KUKA KRL data list: Modul.dat

&ACCESS RVP
&REL 14
DEFDAT Modul PUBLIC
;FOLD EXTERNAL DECLARATIONS;%{PE}%MKUKATPBASIS,%CEXT,%VCOMMON,%P
;FOLD BASISTECH EXT;%{PE}%MKUKATPBASIS,%CEXT,%VEXT,%P
EXT  BAS (BAS_COMMAND  :IN,REAL  :IN )
DECL INT SUCCESS
;ENDFOLD (BASISTECH EXT)
;FOLD USER EXT;%{E}%MKUKATPUSER,%CEXT,%VEXT,%P
;Make here your modifications

;ENDFOLD (USER EXT)
;ENDFOLD (EXTERNAL DECLERATIONS)


DECL E6POS POSITION[4]
DECL INT I
DECL E6POS Xpozy={X 1232,Y -263,Z 1000,A 0,B 67,C -90}

ENDDAT
